Staubli VAL3: setObjectInUse.pgx

public program setObjectInUse(num x_nIdx)
begin
  // This programs is used to count how many users have accessed
  // to the data of an object in the queue
  //
  // Input param
  //  x_nIdx       : Index of the object in the queue
  //
  // Output param
  //  none
  //
  // Created 25-09-07                                   C.CURRIVAND
  //----------------------------------------------------------------
  //
  nNumbOfUser[x_nIdx]=nNumbOfUser[x_nIdx]+1
end
